FUNCTION F_SysTimeToString : STRING(23)
VAR_INPUT
	nSysTime : LINT;
END_VAR
VAR
	nFileTime : T_FILETIME;
	
	fbGetSystemTime  : GETSYSTEMTIME;
END_VAR

MEMCPY(ADR(nFileTime), ADR(nSysTime), SIZEOF(nFileTime));


//F_SysTimeToString := DCTIME64_TO_STRING(FILETIME_TO_DCTIME64(nFileTime));


fbGetSystemTime(timeLoDW=>nFileTime.dwLowDateTime, timeHiDW=>nFileTime.dwHighDateTime );
F_SysTimeToString := SYSTEMTIME_TO_STRING( FILETIME_TO_SYSTEMTIME( nFileTime ) );

END_FUNCTION

(* stored: Version 1.1.0.1, ProductVersion 3.1.4024.12
   POU F_SysTimeToString: Id {d3adb578-3d6c-4cf8-93a2-495357faec0a}, SpecialFunc None *)
